SYSTEM CODEC_TEST (* Data Encoding/Decoding Test *)
  (* Standard: 61499 Feasibility Demo *)
  (* Version 0.9, 2006-03-04, JHC, Holobloc Inc, Adjusted frame sizes for Windows XP. *)
  (* Version 0.8, 2006-03-02, JHC, Holobloc Inc, Inserted delay in MONITOR initialization. *)
  (* Version 0.7, 2004-08-04, JHC, Rockwell Automation, Adjusted field sizes for Swing components. *)
  (* Version 0.6, 2001-06-01, JHC, Rockwell Automation, Changed to new IN_ANY, OUT_ANY. *)
  (* Version 0.5, 2001-05-24, JHC, Rockwell Automation, Added applications. *)
  (* Version 0.4, 2001-05-23, JHC, Rockwell Automation, Corrected UDP addresses *)
  (* Version 0.3, 2001-05-18, JHC, Rockwell Automation, Adjusted layouts *)
  (* Version 0.2, 2000-12-09, JHC, Rockwell Automation, Adjusted window heights *)
  (* Version 0.1, 2000-05-16, JHC, Rockwell Automation, File type changed to ".sys" *)
  (* Version 0.0, 2000-04-21, JHC, Rockwell Automation *)
  APPLICATION TEST_BITS (* Test bit string data types *)
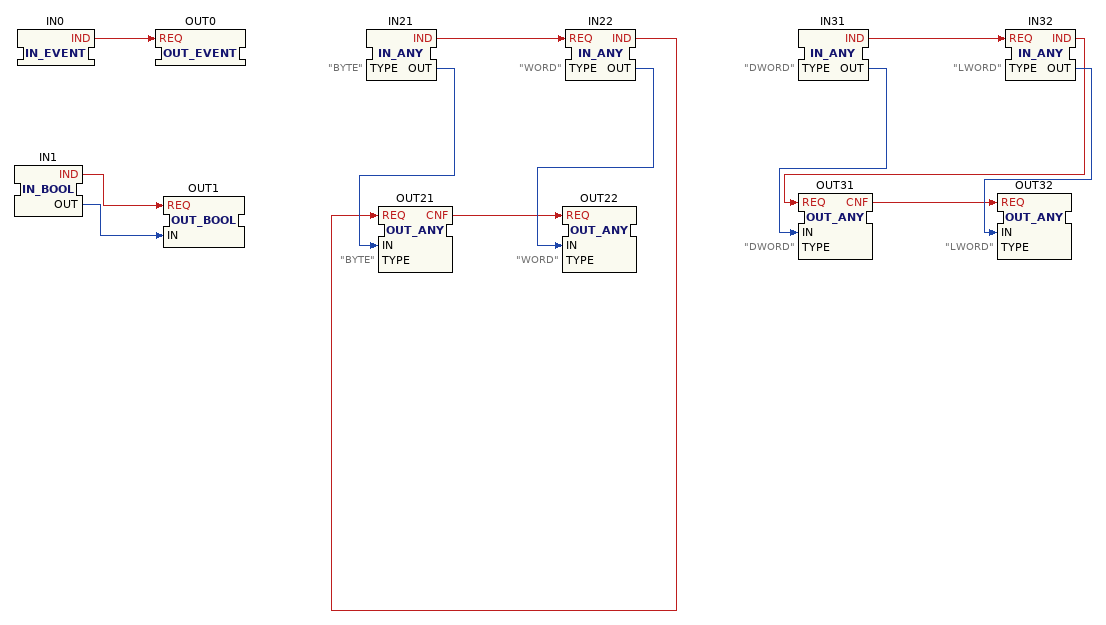
    FBS
      IN0 : IN_EVENT;
      OUT0 : OUT_EVENT;
      IN1 : IN_BOOL;
      OUT1 : OUT_BOOL;
      IN21 : IN_ANY(TYPE := "BYTE");
      OUT21 : OUT_ANY(TYPE := "BYTE");
      IN22 : IN_ANY(TYPE := "WORD");
      OUT22 : OUT_ANY(TYPE := "WORD");
      IN31 : IN_ANY(TYPE := "DWORD");
      OUT31 : OUT_ANY(TYPE := "DWORD");
      IN32 : IN_ANY(TYPE := "LWORD");
      OUT32 : OUT_ANY(TYPE := "LWORD");
    END_FBS
    EVENT_CONNECTIONS
      IN0.IND TO OUT0.REQ;
      IN1.IND TO OUT1.REQ;
      IN21.IND TO IN22.REQ;
      IN22.IND TO OUT21.REQ;
      OUT21.CNF TO OUT22.REQ;
      IN31.IND TO IN32.REQ;
      IN32.IND TO OUT31.REQ;
      OUT31.CNF TO OUT32.REQ;
    END_CONNECTIONS
    DATA_CONNECTIONS
      IN1.OUT TO OUT1.IN;
      IN21.OUT TO OUT21.IN;
      IN22.OUT TO OUT22.IN;
      IN31.OUT TO OUT31.IN;
      IN32.OUT TO OUT32.IN;
    END_CONNECTIONS
  END_APPLICATION
  APPLICATION TEST_INTS (* Test integer data types *)
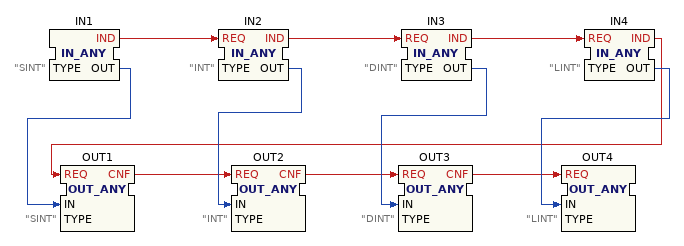
    FBS
      IN1 : IN_ANY(TYPE := "SINT");
      IN2 : IN_ANY(TYPE := "INT");
      IN3 : IN_ANY(TYPE := "DINT");
      IN4 : IN_ANY(TYPE := "LINT");
      OUT1 : OUT_ANY(TYPE := "SINT");
      OUT2 : OUT_ANY(TYPE := "INT");
      OUT3 : OUT_ANY(TYPE := "DINT");
      OUT4 : OUT_ANY(TYPE := "LINT");
    END_FBS
    EVENT_CONNECTIONS
      IN1.IND TO IN2.REQ;
      IN2.IND TO IN3.REQ;
      IN3.IND TO IN4.REQ;
      IN4.IND TO OUT1.REQ;
      OUT1.CNF TO OUT2.REQ;
      OUT2.CNF TO OUT3.REQ;
      OUT3.CNF TO OUT4.REQ;
    END_CONNECTIONS
    DATA_CONNECTIONS
      IN1.OUT TO OUT1.IN;
      IN2.OUT TO OUT2.IN;
      IN3.OUT TO OUT3.IN;
      IN4.OUT TO OUT4.IN;
    END_CONNECTIONS
  END_APPLICATION
  APPLICATION TEST_UINTS (* Test unsigned integer data types *)
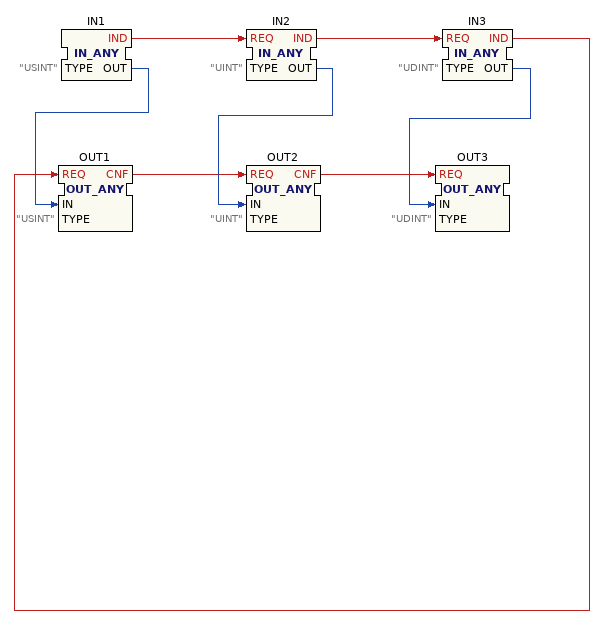
    FBS
      IN1 : IN_ANY(TYPE := "USINT");
      IN2 : IN_ANY(TYPE := "UINT");
      IN3 : IN_ANY(TYPE := "UDINT");
      OUT1 : OUT_ANY(TYPE := "USINT");
      OUT2 : OUT_ANY(TYPE := "UINT");
      OUT3 : OUT_ANY(TYPE := "UDINT");
    END_FBS
    EVENT_CONNECTIONS
      IN1.IND TO IN2.REQ;
      IN2.IND TO IN3.REQ;
      IN3.IND TO OUT1.REQ;
      OUT1.CNF TO OUT2.REQ;
      OUT2.CNF TO OUT3.REQ;
    END_CONNECTIONS
    DATA_CONNECTIONS
      IN1.OUT TO OUT1.IN;
      IN2.OUT TO OUT2.IN;
      IN3.OUT TO OUT3.IN;
    END_CONNECTIONS
  END_APPLICATION
  APPLICATION TEST_REALS (* Test floating point data types *)
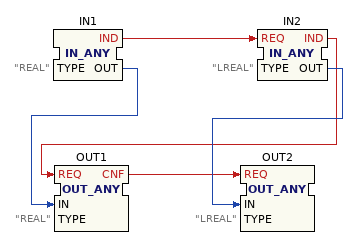
    FBS
      IN1 : IN_ANY(TYPE := "REAL");
      IN2 : IN_ANY(TYPE := "LREAL");
      OUT1 : OUT_ANY(TYPE := "REAL");
      OUT2 : OUT_ANY(TYPE := "LREAL");
    END_FBS
    EVENT_CONNECTIONS
      IN1.IND TO IN2.REQ;
      IN2.IND TO OUT1.REQ;
      OUT1.CNF TO OUT2.REQ;
    END_CONNECTIONS
    DATA_CONNECTIONS
      IN1.OUT TO OUT1.IN;
      IN2.OUT TO OUT2.IN;
    END_CONNECTIONS
  END_APPLICATION
  APPLICATION TEST_TIMES (* Test time data types *)
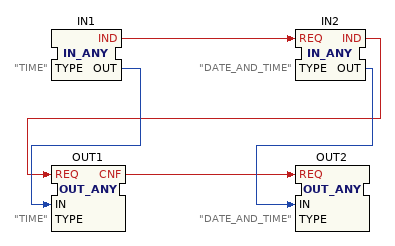
    FBS
      IN1 : IN_ANY(TYPE := "TIME");
      IN2 : IN_ANY(TYPE := "DATE_AND_TIME");
      OUT1 : OUT_ANY(TYPE := "TIME");
      OUT2 : OUT_ANY(TYPE := "DATE_AND_TIME");
    END_FBS
    EVENT_CONNECTIONS
      IN1.IND TO IN2.REQ;
      IN2.IND TO OUT1.REQ;
      OUT1.CNF TO OUT2.REQ;
    END_CONNECTIONS
    DATA_CONNECTIONS
      IN1.OUT TO OUT1.IN;
      IN2.OUT TO OUT2.IN;
    END_CONNECTIONS
  END_APPLICATION
  APPLICATION TEST_STRINGS (* Test string data types *)
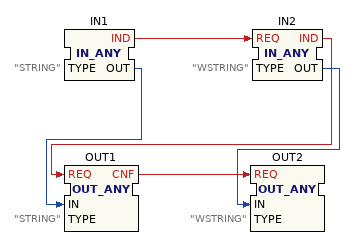
    FBS
      IN1 : IN_ANY(TYPE := "STRING");
      IN2 : IN_ANY(TYPE := "WSTRING");
      OUT1 : OUT_ANY(TYPE := "STRING");
      OUT2 : OUT_ANY(TYPE := "WSTRING");
    END_FBS
    EVENT_CONNECTIONS
      IN1.IND TO IN2.REQ;
      IN2.IND TO OUT1.REQ;
      OUT1.CNF TO OUT2.REQ;
    END_CONNECTIONS
    DATA_CONNECTIONS
      IN1.OUT TO OUT1.IN;
      IN2.OUT TO OUT2.IN;
    END_CONNECTIONS
  END_APPLICATION
  APPLICATION TEST_ARRAY (* Test ARRAYs *)
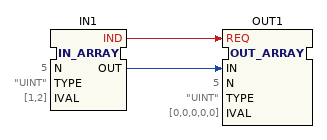
    FBS
      IN1 : IN_ARRAY(N := 5, TYPE := "UINT", IVAL := [1,2]);
      OUT1 : OUT_ARRAY(N := 5, TYPE := "UINT", IVAL := [0,0,0,0,0]);
    END_FBS
    EVENT_CONNECTIONS
      IN1.IND TO OUT1.REQ;
    END_CONNECTIONS
    DATA_CONNECTIONS
      IN1.OUT TO OUT1.IN;
    END_CONNECTIONS
  END_APPLICATION
  APPLICATION TEST_COLOR (* Test  COLOR - Just for fun! *)
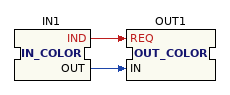
    FBS
      IN1 : IN_COLOR;
      OUT1 : OUT_COLOR;
    END_FBS
    EVENT_CONNECTIONS
      IN1.IND TO OUT1.REQ;
    END_CONNECTIONS
    DATA_CONNECTIONS
      IN1.OUT TO OUT1.IN;
    END_CONNECTIONS
  END_APPLICATION
  DEVICE SEND_BITS : FRAME_DEVICE(BOUNDS := [50,50,175,195], GRID := [1,1])
    RESOURCE RES0 : PANEL_RESOURCE
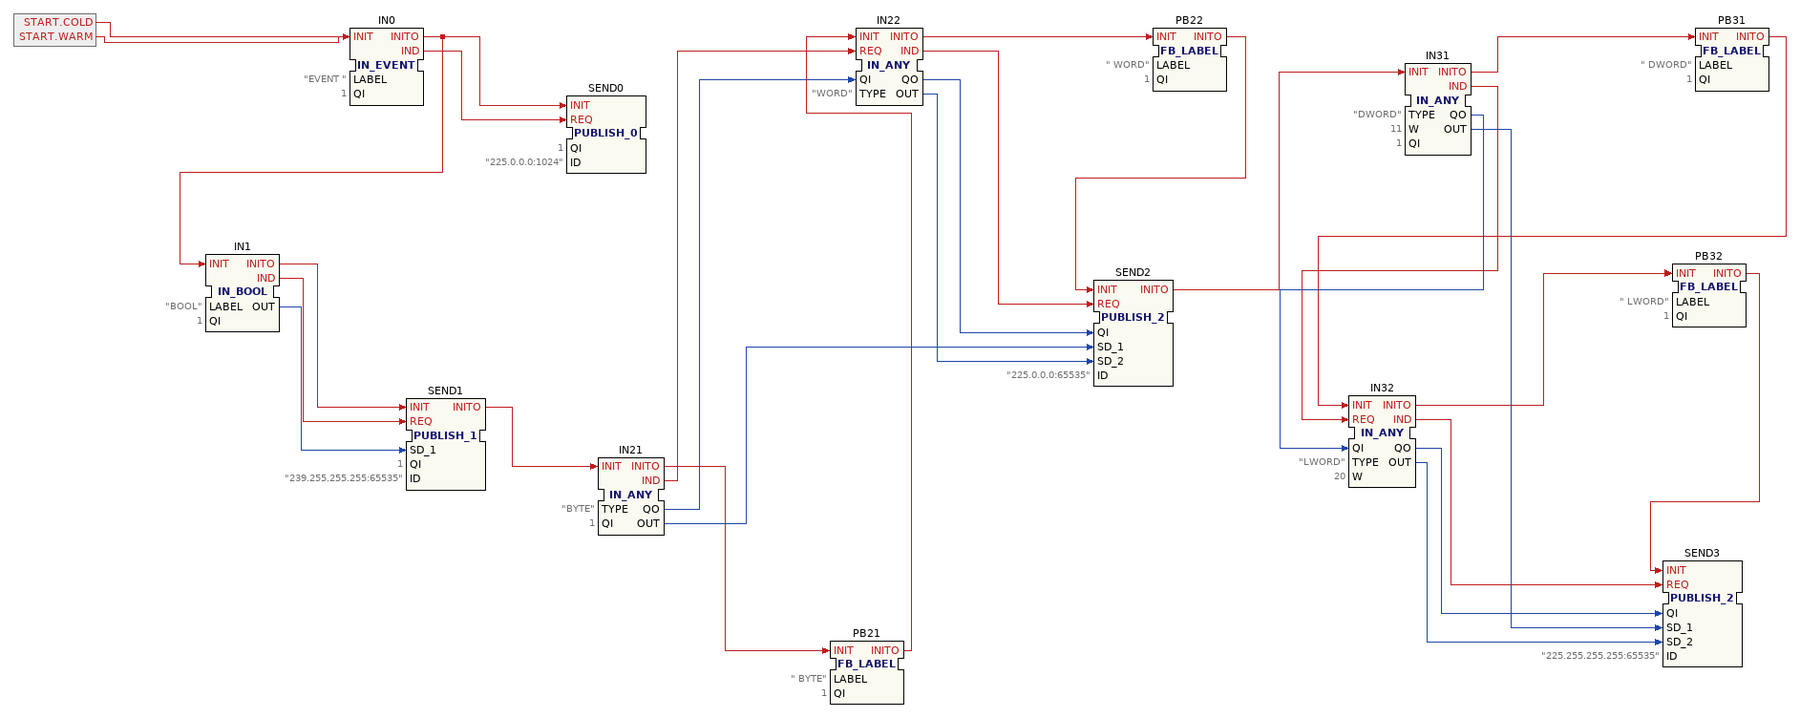
      FBS
        IN0 : IN_EVENT(LABEL := "EVENT   ", QI := 1);
        SEND0 : PUBLISH_0(QI := 1, ID := "225.0.0.0:1024");
        IN1 : IN_BOOL(LABEL := "BOOL", QI := 1);
        SEND1 : PUBLISH_1(QI := 1, ID := "239.255.255.255:65535");
        PB21 : FB_LABEL(LABEL := " BYTE", QI := 1);
        IN21 : IN_ANY(TYPE := "BYTE", QI := 1);
        PB22 : FB_LABEL(LABEL := " WORD", QI := 1);
        IN22 : IN_ANY(TYPE := "WORD");
        SEND2 : PUBLISH_2(ID := "225.0.0.0:65535");
        PB31 : FB_LABEL(LABEL := " DWORD", QI := 1);
        IN31 : IN_ANY(TYPE := "DWORD", W := 11, QI := 1);
        PB32 : FB_LABEL(LABEL := " LWORD", QI := 1);
        IN32 : IN_ANY(TYPE := "LWORD", W := 20);
        SEND3 : PUBLISH_2(ID := "225.255.255.255:65535");
      END_FBS
      EVENT_CONNECTIONS
        START.COLD TO IN0.INIT;
        START.WARM TO IN0.INIT;
        IN0.INITO TO SEND0.INIT;
        IN0.INITO TO IN1.INIT;
        IN1.INITO TO SEND1.INIT;
        SEND1.INITO TO IN21.INIT;
        IN21.INITO TO PB21.INIT;
        PB21.INITO TO IN22.INIT;
        IN22.INITO TO PB22.INIT;
        PB22.INITO TO SEND2.INIT;
        SEND2.INITO TO IN31.INIT;
        IN31.INITO TO PB31.INIT;
        PB31.INITO TO IN32.INIT;
        IN32.INITO TO PB32.INIT;
        PB32.INITO TO SEND3.INIT;
        IN0.IND TO SEND0.REQ;
        IN1.IND TO SEND1.REQ;
        IN21.IND TO IN22.REQ;
        IN22.IND TO SEND2.REQ;
        IN31.IND TO IN32.REQ;
        IN32.IND TO SEND3.REQ;
      END_CONNECTIONS
      DATA_CONNECTIONS
        IN21.QO TO IN22.QI;
        IN22.QO TO SEND2.QI;
        IN31.QO TO IN32.QI;
        IN32.QO TO SEND3.QI;
        IN1.OUT TO SEND1.SD_1;
        IN21.OUT TO SEND2.SD_1;
        IN22.OUT TO SEND2.SD_2;
        IN31.OUT TO SEND3.SD_1;
        IN32.OUT TO SEND3.SD_2;
      END_CONNECTIONS
    END_RESOURCE
  END_DEVICE
  DEVICE RCV_BITS : FRAME_DEVICE(BOUNDS := [225,50,175,195], GRID := [1,1])
    RESOURCE RES0 : PANEL_RESOURCE
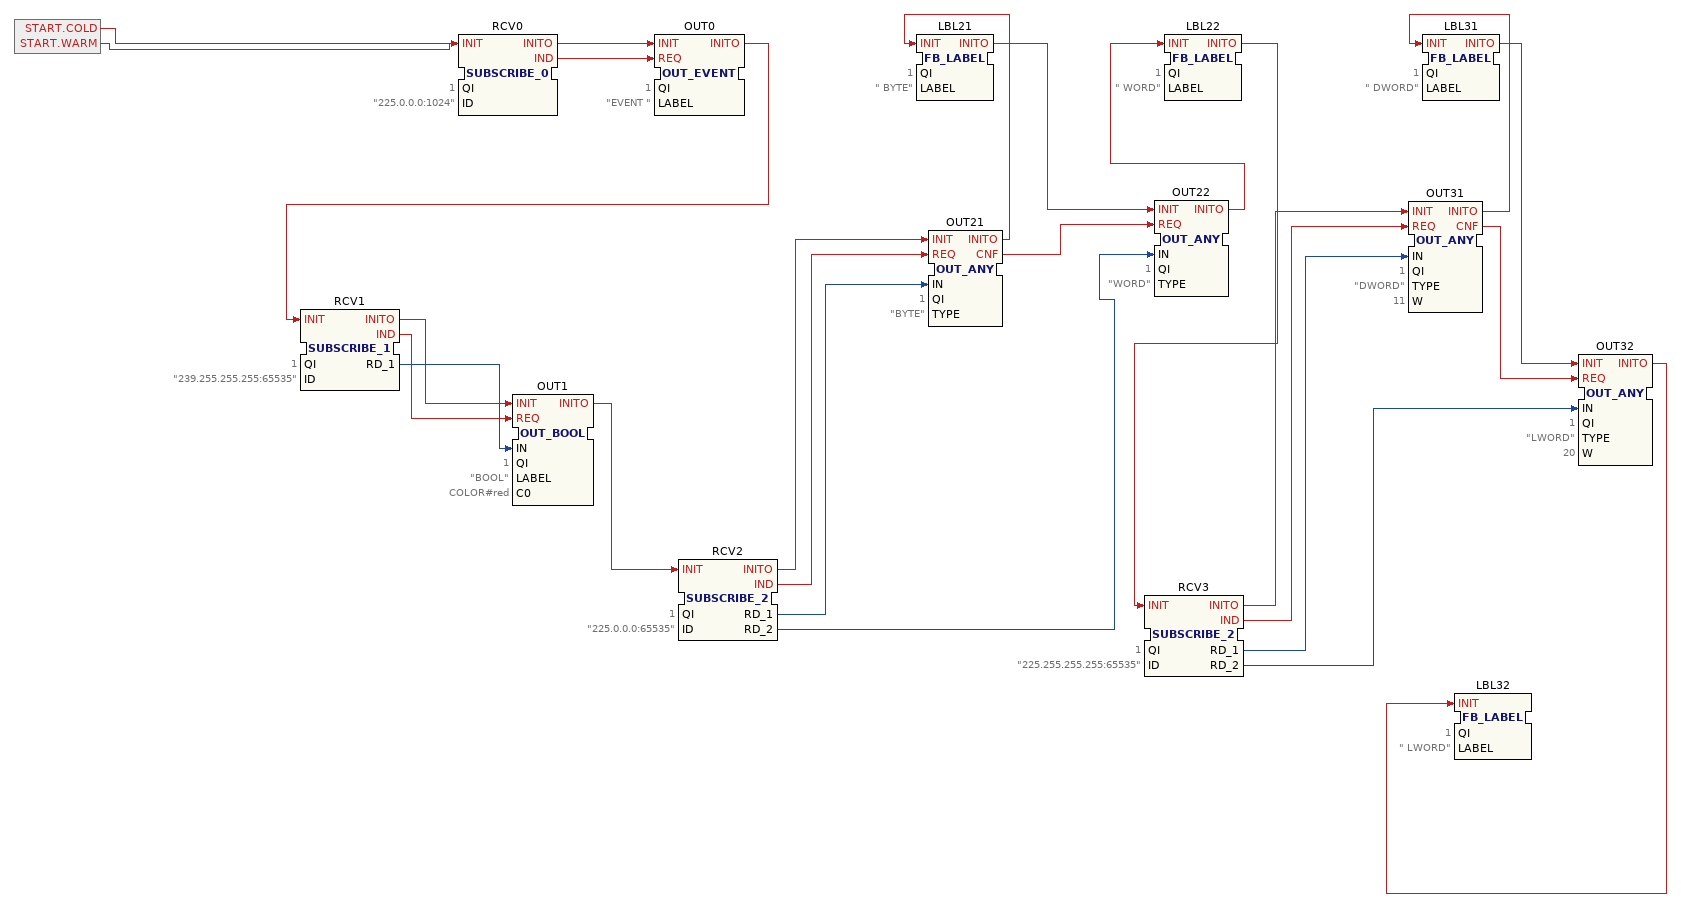
      FBS
        RCV0 : SUBSCRIBE_0(QI := 1, ID := "225.0.0.0:1024");
        OUT0 : OUT_EVENT(QI := 1, LABEL := "EVENT   ");
        RCV1 : SUBSCRIBE_1(QI := 1, ID := "239.255.255.255:65535");
        OUT1 : OUT_BOOL(QI := 1, LABEL := "BOOL", C0 := COLOR#red);
        RCV2 : SUBSCRIBE_2(QI := 1, ID := "225.0.0.0:65535");
        LBL21 : FB_LABEL(QI := 1, LABEL := " BYTE");
        OUT21 : OUT_ANY(QI := 1, TYPE := "BYTE");
        LBL22 : FB_LABEL(QI := 1, LABEL := " WORD");
        OUT22 : OUT_ANY(QI := 1, TYPE := "WORD");
        RCV3 : SUBSCRIBE_2(QI := 1, ID := "225.255.255.255:65535");
        LBL31 : FB_LABEL(QI := 1, LABEL := " DWORD");
        OUT31 : OUT_ANY(QI := 1, TYPE := "DWORD", W := 11);
        LBL32 : FB_LABEL(QI := 1, LABEL := " LWORD");
        OUT32 : OUT_ANY(QI := 1, TYPE := "LWORD", W := 20);
      END_FBS
      EVENT_CONNECTIONS
        START.COLD TO RCV0.INIT;
        START.WARM TO RCV0.INIT;
        RCV0.INITO TO OUT0.INIT;
        OUT0.INITO TO RCV1.INIT;
        RCV1.INITO TO OUT1.INIT;
        OUT1.INITO TO RCV2.INIT;
        RCV2.INITO TO OUT21.INIT;
        OUT21.INITO TO LBL21.INIT;
        LBL21.INITO TO OUT22.INIT;
        OUT22.INITO TO LBL22.INIT;
        LBL22.INITO TO RCV3.INIT;
        RCV3.INITO TO OUT31.INIT;
        OUT31.INITO TO LBL31.INIT;
        LBL31.INITO TO OUT32.INIT;
        OUT32.INITO TO LBL32.INIT;
        RCV0.IND TO OUT0.REQ;
        RCV1.IND TO OUT1.REQ;
        RCV2.IND TO OUT21.REQ;
        OUT21.CNF TO OUT22.REQ;
        RCV3.IND TO OUT31.REQ;
        OUT31.CNF TO OUT32.REQ;
      END_CONNECTIONS
      DATA_CONNECTIONS
        RCV1.RD_1 TO OUT1.IN;
        RCV2.RD_1 TO OUT21.IN;
        RCV2.RD_2 TO OUT22.IN;
        RCV3.RD_1 TO OUT31.IN;
        RCV3.RD_2 TO OUT32.IN;
      END_CONNECTIONS
    END_RESOURCE
  END_DEVICE
  DEVICE SEND_INTS : FRAME_DEVICE(BOUNDS := [50,240,175,170], GRID := [1,1])
    RESOURCE RES0 : PANEL_RESOURCE
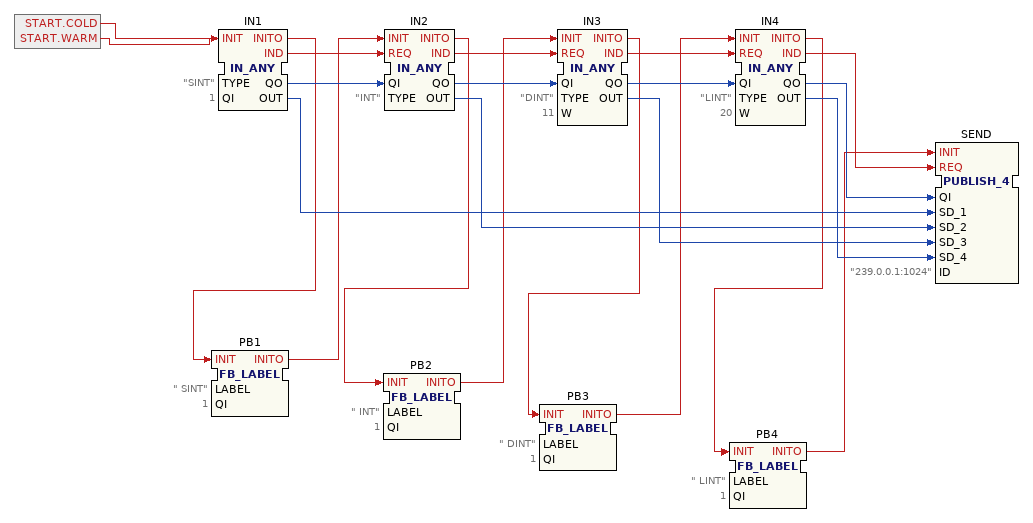
      FBS
        PB1 : FB_LABEL(LABEL := " SINT", QI := 1);
        IN1 : IN_ANY(TYPE := "SINT", QI := 1);
        PB2 : FB_LABEL(LABEL := " INT", QI := 1);
        IN2 : IN_ANY(TYPE := "INT");
        PB3 : FB_LABEL(LABEL := " DINT", QI := 1);
        IN3 : IN_ANY(TYPE := "DINT", W := 11);
        PB4 : FB_LABEL(LABEL := " LINT", QI := 1);
        IN4 : IN_ANY(TYPE := "LINT", W := 20);
        SEND : PUBLISH_4(ID := "239.0.0.1:1024");
      END_FBS
      EVENT_CONNECTIONS
        START.COLD TO IN1.INIT;
        START.WARM TO IN1.INIT;
        IN1.INITO TO PB1.INIT;
        PB1.INITO TO IN2.INIT;
        IN2.INITO TO PB2.INIT;
        PB2.INITO TO IN3.INIT;
        IN3.INITO TO PB3.INIT;
        PB3.INITO TO IN4.INIT;
        IN4.INITO TO PB4.INIT;
        PB4.INITO TO SEND.INIT;
        IN1.IND TO IN2.REQ;
        IN2.IND TO IN3.REQ;
        IN3.IND TO IN4.REQ;
        IN4.IND TO SEND.REQ;
      END_CONNECTIONS
      DATA_CONNECTIONS
        IN1.QO TO IN2.QI;
        IN2.QO TO IN3.QI;
        IN3.QO TO IN4.QI;
        IN4.QO TO SEND.QI;
        IN1.OUT TO SEND.SD_1;
        IN2.OUT TO SEND.SD_2;
        IN3.OUT TO SEND.SD_3;
        IN4.OUT TO SEND.SD_4;
      END_CONNECTIONS
    END_RESOURCE
  END_DEVICE
  DEVICE RCV_INTS : FRAME_DEVICE(BOUNDS := [225,240,175,170], GRID := [1,1])
    RESOURCE RES0 : PANEL_RESOURCE
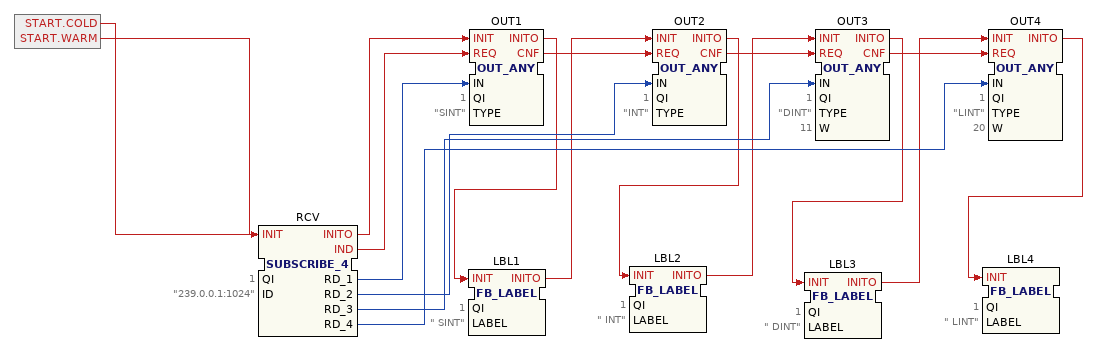
      FBS
        RCV : SUBSCRIBE_4(QI := 1, ID := "239.0.0.1:1024");
        LBL1 : FB_LABEL(QI := 1, LABEL := " SINT");
        OUT1 : OUT_ANY(QI := 1, TYPE := "SINT");
        LBL2 : FB_LABEL(QI := 1, LABEL := " INT");
        OUT2 : OUT_ANY(QI := 1, TYPE := "INT");
        LBL3 : FB_LABEL(QI := 1, LABEL := " DINT");
        OUT3 : OUT_ANY(QI := 1, TYPE := "DINT", W := 11);
        LBL4 : FB_LABEL(QI := 1, LABEL := " LINT");
        OUT4 : OUT_ANY(QI := 1, TYPE := "LINT", W := 20);
      END_FBS
      EVENT_CONNECTIONS
        START.COLD TO RCV.INIT;
        START.WARM TO RCV.INIT;
        RCV.INITO TO OUT1.INIT;
        OUT1.INITO TO LBL1.INIT;
        LBL1.INITO TO OUT2.INIT;
        OUT2.INITO TO LBL2.INIT;
        LBL2.INITO TO OUT3.INIT;
        OUT3.INITO TO LBL3.INIT;
        LBL3.INITO TO OUT4.INIT;
        OUT4.INITO TO LBL4.INIT;
        RCV.IND TO OUT1.REQ;
        OUT1.CNF TO OUT2.REQ;
        OUT2.CNF TO OUT3.REQ;
        OUT3.CNF TO OUT4.REQ;
      END_CONNECTIONS
      DATA_CONNECTIONS
        RCV.RD_1 TO OUT1.IN;
        RCV.RD_2 TO OUT2.IN;
        RCV.RD_3 TO OUT3.IN;
        RCV.RD_4 TO OUT4.IN;
      END_CONNECTIONS
    END_RESOURCE
  END_DEVICE
  DEVICE SEND_UINTS : FRAME_DEVICE(BOUNDS := [50,405,175,120], GRID := [1,1])
    RESOURCE RES0 : PANEL_RESOURCE
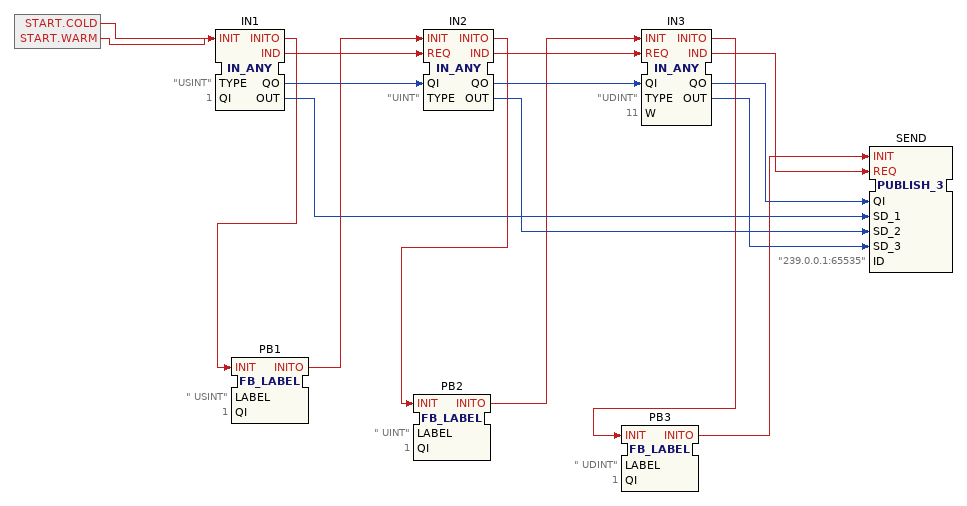
      FBS
        PB1 : FB_LABEL(LABEL := " USINT", QI := 1);
        IN1 : IN_ANY(TYPE := "USINT", QI := 1);
        PB2 : FB_LABEL(LABEL := " UINT", QI := 1);
        IN2 : IN_ANY(TYPE := "UINT");
        PB3 : FB_LABEL(LABEL := " UDINT", QI := 1);
        IN3 : IN_ANY(TYPE := "UDINT", W := 11);
        SEND : PUBLISH_3(ID := "239.0.0.1:65535");
      END_FBS
      EVENT_CONNECTIONS
        START.COLD TO IN1.INIT;
        START.WARM TO IN1.INIT;
        IN1.INITO TO PB1.INIT;
        PB1.INITO TO IN2.INIT;
        IN2.INITO TO PB2.INIT;
        PB2.INITO TO IN3.INIT;
        IN3.INITO TO PB3.INIT;
        PB3.INITO TO SEND.INIT;
        IN1.IND TO IN2.REQ;
        IN2.IND TO IN3.REQ;
        IN3.IND TO SEND.REQ;
      END_CONNECTIONS
      DATA_CONNECTIONS
        IN1.QO TO IN2.QI;
        IN2.QO TO IN3.QI;
        IN3.QO TO SEND.QI;
        IN1.OUT TO SEND.SD_1;
        IN2.OUT TO SEND.SD_2;
        IN3.OUT TO SEND.SD_3;
      END_CONNECTIONS
    END_RESOURCE
  END_DEVICE
  DEVICE RCV_UINTS : FRAME_DEVICE(BOUNDS := [225,405,175,120], GRID := [1,1])
    RESOURCE RES0 : PANEL_RESOURCE
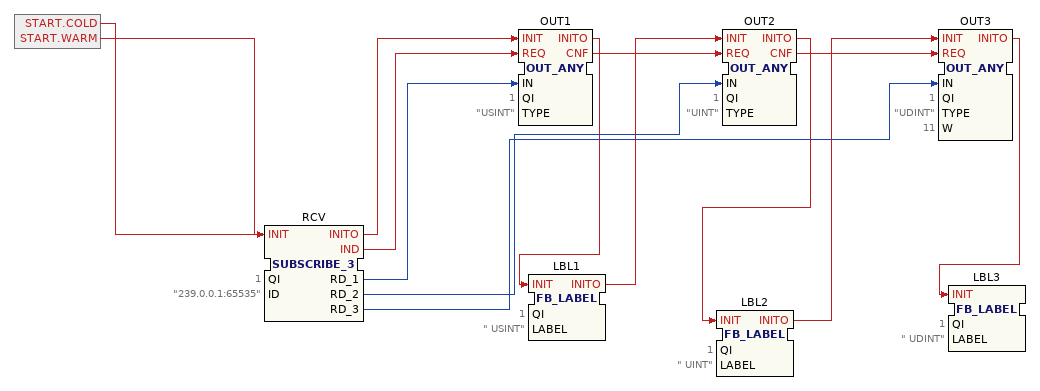
      FBS
        RCV : SUBSCRIBE_3(QI := 1, ID := "239.0.0.1:65535");
        LBL1 : FB_LABEL(QI := 1, LABEL := " USINT");
        OUT1 : OUT_ANY(QI := 1, TYPE := "USINT");
        LBL2 : FB_LABEL(QI := 1, LABEL := " UINT");
        OUT2 : OUT_ANY(QI := 1, TYPE := "UINT");
        LBL3 : FB_LABEL(QI := 1, LABEL := " UDINT");
        OUT3 : OUT_ANY(QI := 1, TYPE := "UDINT", W := 11);
      END_FBS
      EVENT_CONNECTIONS
        START.COLD TO RCV.INIT;
        START.WARM TO RCV.INIT;
        RCV.INITO TO OUT1.INIT;
        OUT1.INITO TO LBL1.INIT;
        LBL1.INITO TO OUT2.INIT;
        OUT2.INITO TO LBL2.INIT;
        LBL2.INITO TO OUT3.INIT;
        OUT3.INITO TO LBL3.INIT;
        RCV.IND TO OUT1.REQ;
        OUT1.CNF TO OUT2.REQ;
        OUT2.CNF TO OUT3.REQ;
      END_CONNECTIONS
      DATA_CONNECTIONS
        RCV.RD_1 TO OUT1.IN;
        RCV.RD_2 TO OUT2.IN;
        RCV.RD_3 TO OUT3.IN;
      END_CONNECTIONS
    END_RESOURCE
  END_DEVICE
  DEVICE SEND_REALS : FRAME_DEVICE(BOUNDS := [50,520,175,100], GRID := [1,1])
    RESOURCE RES0 : PANEL_RESOURCE
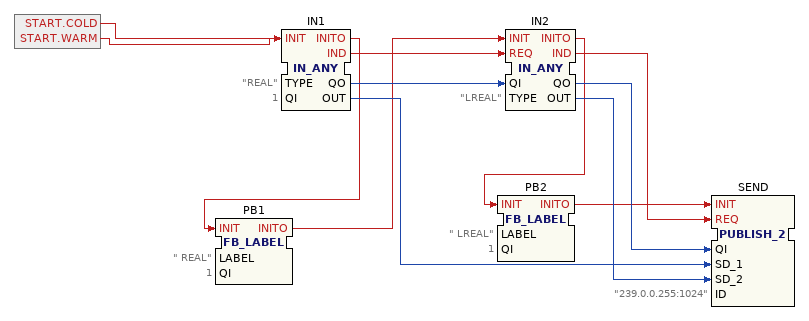
      FBS
        PB1 : FB_LABEL(LABEL := " REAL", QI := 1);
        IN1 : IN_ANY(TYPE := "REAL", QI := 1);
        PB2 : FB_LABEL(LABEL := " LREAL", QI := 1);
        IN2 : IN_ANY(TYPE := "LREAL");
        SEND : PUBLISH_2(ID := "239.0.0.255:1024");
      END_FBS
      EVENT_CONNECTIONS
        START.COLD TO IN1.INIT;
        START.WARM TO IN1.INIT;
        IN1.INITO TO PB1.INIT;
        PB1.INITO TO IN2.INIT;
        IN2.INITO TO PB2.INIT;
        PB2.INITO TO SEND.INIT;
        IN1.IND TO IN2.REQ;
        IN2.IND TO SEND.REQ;
      END_CONNECTIONS
      DATA_CONNECTIONS
        IN1.QO TO IN2.QI;
        IN2.QO TO SEND.QI;
        IN1.OUT TO SEND.SD_1;
        IN2.OUT TO SEND.SD_2;
      END_CONNECTIONS
    END_RESOURCE
  END_DEVICE
  DEVICE RCV_REALS : FRAME_DEVICE(BOUNDS := [225,520,175,100], GRID := [1,1])
    RESOURCE RES0 : PANEL_RESOURCE
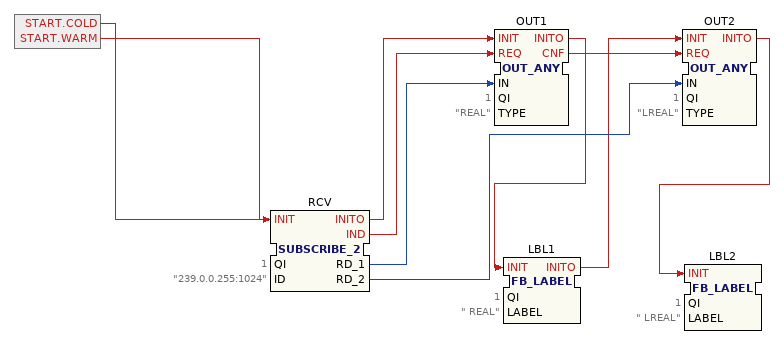
      FBS
        RCV : SUBSCRIBE_2(QI := 1, ID := "239.0.0.255:1024");
        LBL1 : FB_LABEL(QI := 1, LABEL := " REAL");
        OUT1 : OUT_ANY(QI := 1, TYPE := "REAL");
        LBL2 : FB_LABEL(QI := 1, LABEL := " LREAL");
        OUT2 : OUT_ANY(QI := 1, TYPE := "LREAL");
      END_FBS
      EVENT_CONNECTIONS
        START.COLD TO RCV.INIT;
        START.WARM TO RCV.INIT;
        RCV.INITO TO OUT1.INIT;
        OUT1.INITO TO LBL1.INIT;
        LBL1.INITO TO OUT2.INIT;
        OUT2.INITO TO LBL2.INIT;
        RCV.IND TO OUT1.REQ;
        OUT1.CNF TO OUT2.REQ;
      END_CONNECTIONS
      DATA_CONNECTIONS
        RCV.RD_1 TO OUT1.IN;
        RCV.RD_2 TO OUT2.IN;
      END_CONNECTIONS
    END_RESOURCE
  END_DEVICE
  DEVICE MONITOR : FRAME_DEVICE(BOUNDS := [400,50,400,225], GRID := [1,1])
    RESOURCE RES0 : PANEL_RESOURCE
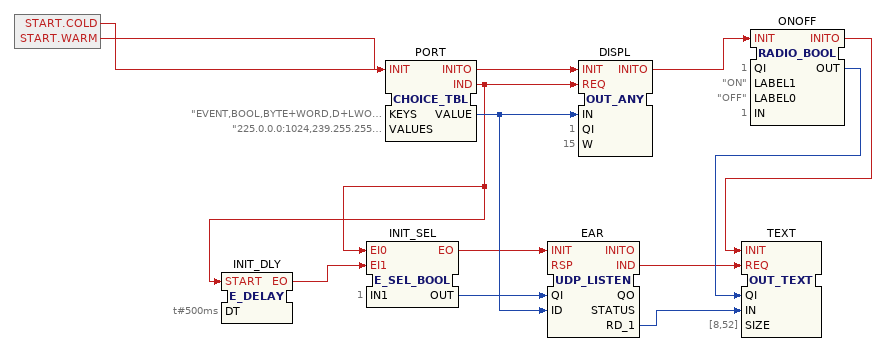
      FBS
        PORT : CHOICE_TBL(KEYS := "EVENT,BOOL,BYTE+WORD,D+LWORD,INTS,UINTS,REALS,TIMES,STRINGS,ARRAYS,COLOR", VALUES := "225.0.0.0:1024,239.255.255.255:65535,225.0.0.0:65535,225.255.255.255:65535,239.0.0.1:1024,239.0.0.1:65535,239.0.0.255:1024,239.0.0.255:65535,239.0.255.255:1024,239.0.255.255:65535,239.255.255.255:1024");
        DISPL : OUT_ANY(QI := 1, W := 15);
        EAR : UDP_LISTEN;
        ONOFF : RADIO_BOOL(QI := 1, LABEL1 := "ON", LABEL0 := "OFF", IN := 1);
        TEXT : OUT_TEXT(SIZE := [8,52]);
        INIT_SEL : E_SEL_BOOL(IN1 := 1);
        INIT_DLY : E_DELAY(DT := t#500ms);
      END_FBS
      EVENT_CONNECTIONS
        START.COLD TO PORT.INIT;
        START.WARM TO PORT.INIT;
        PORT.INITO TO DISPL.INIT;
        DISPL.INITO TO ONOFF.INIT;
        ONOFF.INITO TO TEXT.INIT;
        PORT.IND TO DISPL.REQ;
        EAR.IND TO TEXT.REQ;
        PORT.IND TO INIT_SEL.EI0;
        INIT_SEL.EO TO EAR.INIT;
        INIT_DLY.EO TO INIT_SEL.EI1;
        PORT.IND TO INIT_DLY.START;
      END_CONNECTIONS
      DATA_CONNECTIONS
        PORT.VALUE TO DISPL.IN;
        PORT.VALUE TO EAR.ID;
        ONOFF.OUT TO TEXT.QI;
        EAR.RD_1 TO TEXT.IN;
        INIT_SEL.OUT TO EAR.QI;
      END_CONNECTIONS
    END_RESOURCE
  END_DEVICE
  DEVICE SEND_TIMES : FRAME_DEVICE(BOUNDS := [400,270,200,115], GRID := [1,1])
    RESOURCE RES0 : PANEL_RESOURCE
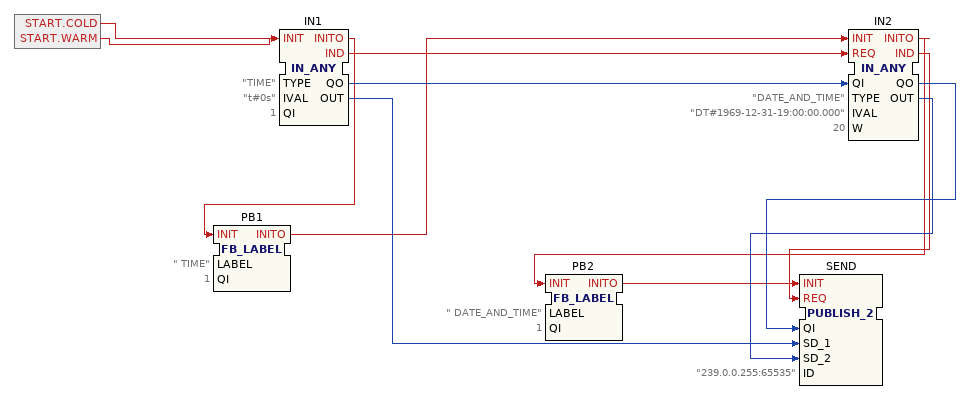
      FBS
        PB1 : FB_LABEL(LABEL := " TIME", QI := 1);
        IN1 : IN_ANY(TYPE := "TIME", IVAL := "t#0s", QI := 1);
        PB2 : FB_LABEL(LABEL := " DATE_AND_TIME", QI := 1);
        IN2 : IN_ANY(TYPE := "DATE_AND_TIME", IVAL := "DT#1969-12-31-19:00:00.000", W := 20);
        SEND : PUBLISH_2(ID := "239.0.0.255:65535");
      END_FBS
      EVENT_CONNECTIONS
        START.COLD TO IN1.INIT;
        START.WARM TO IN1.INIT;
        IN1.INITO TO PB1.INIT;
        PB1.INITO TO IN2.INIT;
        IN2.INITO TO PB2.INIT;
        PB2.INITO TO SEND.INIT;
        IN1.IND TO IN2.REQ;
        IN2.IND TO SEND.REQ;
      END_CONNECTIONS
      DATA_CONNECTIONS
        IN1.QO TO IN2.QI;
        IN2.QO TO SEND.QI;
        IN1.OUT TO SEND.SD_1;
        IN2.OUT TO SEND.SD_2;
      END_CONNECTIONS
    END_RESOURCE
  END_DEVICE
  DEVICE RCV_TIMES : FRAME_DEVICE(BOUNDS := [600,270,200,115], GRID := [1,1])
    RESOURCE RES0 : PANEL_RESOURCE
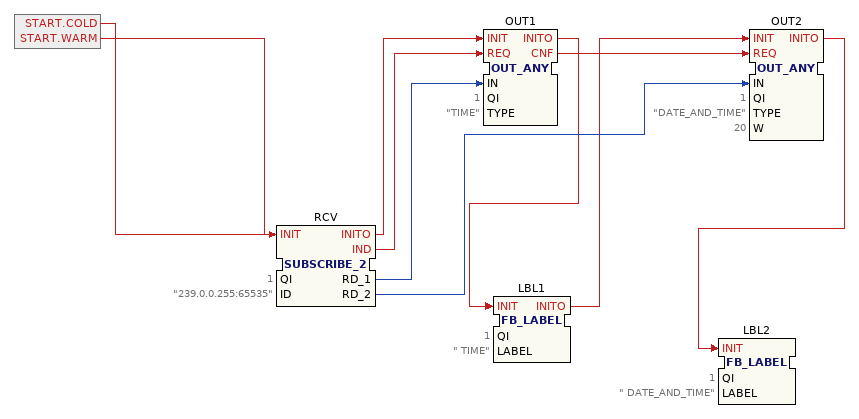
      FBS
        RCV : SUBSCRIBE_2(QI := 1, ID := "239.0.0.255:65535");
        LBL1 : FB_LABEL(QI := 1, LABEL := " TIME");
        OUT1 : OUT_ANY(QI := 1, TYPE := "TIME");
        LBL2 : FB_LABEL(QI := 1, LABEL := " DATE_AND_TIME");
        OUT2 : OUT_ANY(QI := 1, TYPE := "DATE_AND_TIME", W := 20);
      END_FBS
      EVENT_CONNECTIONS
        START.COLD TO RCV.INIT;
        START.WARM TO RCV.INIT;
        RCV.INITO TO OUT1.INIT;
        OUT1.INITO TO LBL1.INIT;
        LBL1.INITO TO OUT2.INIT;
        OUT2.INITO TO LBL2.INIT;
        RCV.IND TO OUT1.REQ;
        OUT1.CNF TO OUT2.REQ;
      END_CONNECTIONS
      DATA_CONNECTIONS
        RCV.RD_1 TO OUT1.IN;
        RCV.RD_2 TO OUT2.IN;
      END_CONNECTIONS
    END_RESOURCE
  END_DEVICE
  DEVICE SEND_STRINGS : FRAME_DEVICE(BOUNDS := [400,385,200,95], GRID := [1,1])
    RESOURCE RES0 : PANEL_RESOURCE
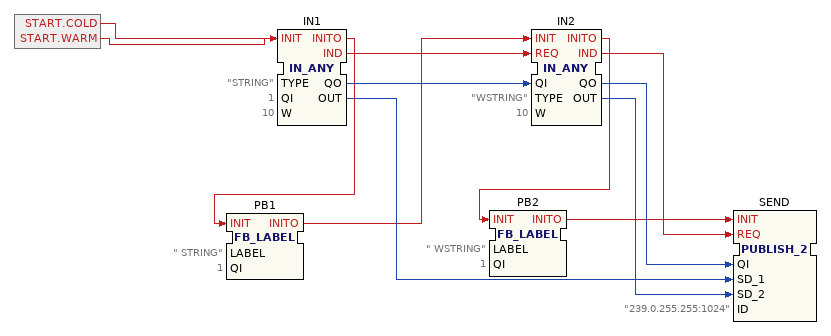
      FBS
        PB1 : FB_LABEL(LABEL := " STRING", QI := 1);
        IN1 : IN_ANY(TYPE := "STRING", QI := 1, W := 10);
        PB2 : FB_LABEL(LABEL := " WSTRING", QI := 1);
        IN2 : IN_ANY(TYPE := "WSTRING", W := 10);
        SEND : PUBLISH_2(ID := "239.0.255.255:1024");
      END_FBS
      EVENT_CONNECTIONS
        START.COLD TO IN1.INIT;
        START.WARM TO IN1.INIT;
        IN1.INITO TO PB1.INIT;
        PB1.INITO TO IN2.INIT;
        IN2.INITO TO PB2.INIT;
        PB2.INITO TO SEND.INIT;
        IN1.IND TO IN2.REQ;
        IN2.IND TO SEND.REQ;
      END_CONNECTIONS
      DATA_CONNECTIONS
        IN1.QO TO IN2.QI;
        IN2.QO TO SEND.QI;
        IN1.OUT TO SEND.SD_1;
        IN2.OUT TO SEND.SD_2;
      END_CONNECTIONS
    END_RESOURCE
  END_DEVICE
  DEVICE RCV_STRINGS : FRAME_DEVICE(BOUNDS := [600,385,200,95], GRID := [1,1])
    RESOURCE RES0 : PANEL_RESOURCE
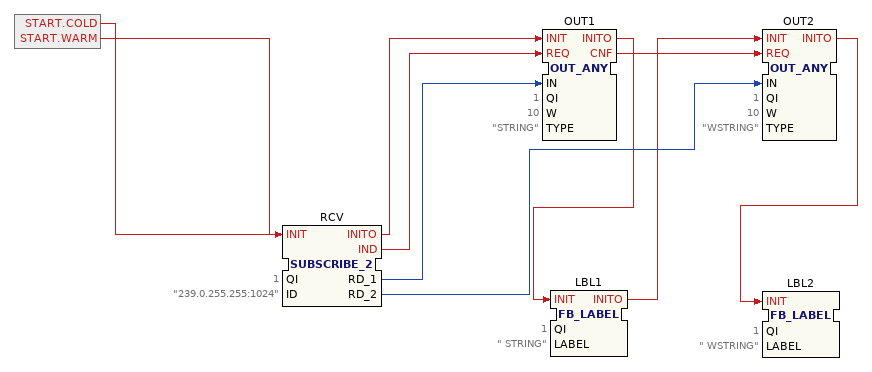
      FBS
        RCV : SUBSCRIBE_2(QI := 1, ID := "239.0.255.255:1024");
        LBL1 : FB_LABEL(QI := 1, LABEL := " STRING");
        OUT1 : OUT_ANY(QI := 1, W := 10, TYPE := "STRING");
        LBL2 : FB_LABEL(QI := 1, LABEL := " WSTRING");
        OUT2 : OUT_ANY(QI := 1, W := 10, TYPE := "WSTRING");
      END_FBS
      EVENT_CONNECTIONS
        START.COLD TO RCV.INIT;
        START.WARM TO RCV.INIT;
        RCV.INITO TO OUT1.INIT;
        OUT1.INITO TO LBL1.INIT;
        LBL1.INITO TO OUT2.INIT;
        OUT2.INITO TO LBL2.INIT;
        RCV.IND TO OUT1.REQ;
        OUT1.CNF TO OUT2.REQ;
      END_CONNECTIONS
      DATA_CONNECTIONS
        RCV.RD_1 TO OUT1.IN;
        RCV.RD_2 TO OUT2.IN;
      END_CONNECTIONS
    END_RESOURCE
  END_DEVICE
  DEVICE SEND_ARRAY : FRAME_DEVICE(BOUNDS := [400,480,210,80], GRID := [1,1])
    RESOURCE RES0 : PANEL_RESOURCE
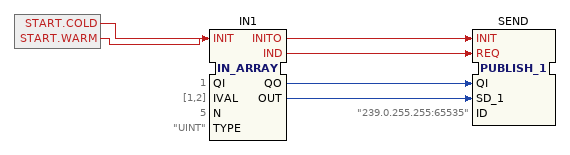
      FBS
        IN1 : IN_ARRAY(QI := 1, IVAL := [1,2], N := 5, TYPE := "UINT");
        SEND : PUBLISH_1(ID := "239.0.255.255:65535");
      END_FBS
      EVENT_CONNECTIONS
        START.COLD TO IN1.INIT;
        START.WARM TO IN1.INIT;
        IN1.INITO TO SEND.INIT;
        IN1.IND TO SEND.REQ;
      END_CONNECTIONS
      DATA_CONNECTIONS
        IN1.QO TO SEND.QI;
        IN1.OUT TO SEND.SD_1;
      END_CONNECTIONS
    END_RESOURCE
  END_DEVICE
  DEVICE RCV_ARRAY : FRAME_DEVICE(BOUNDS := [610,480,190,80], GRID := [1,1])
    RESOURCE RES0 : PANEL_RESOURCE
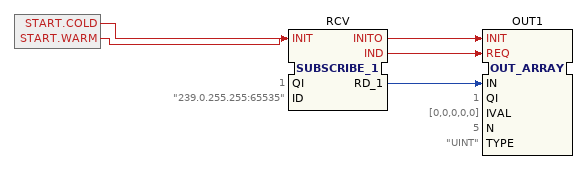
      FBS
        RCV : SUBSCRIBE_1(QI := 1, ID := "239.0.255.255:65535");
        OUT1 : OUT_ARRAY(QI := 1, IVAL := [0,0,0,0,0], N := 5, TYPE := "UINT");
      END_FBS
      EVENT_CONNECTIONS
        START.COLD TO RCV.INIT;
        START.WARM TO RCV.INIT;
        RCV.INITO TO OUT1.INIT;
        RCV.IND TO OUT1.REQ;
      END_CONNECTIONS
      DATA_CONNECTIONS
        RCV.RD_1 TO OUT1.IN;
      END_CONNECTIONS
    END_RESOURCE
  END_DEVICE
  DEVICE SEND_COLOR : FRAME_DEVICE(BOUNDS := [400,560,210,90], GRID := [1,1])
    RESOURCE RES0 : PANEL_RESOURCE
      FBS
        IN1 : IN_COLOR(QI := 1);
        SEND : PUBLISH_1(QI := 1, ID := "239.255.255.255:1024");
      END_FBS
      EVENT_CONNECTIONS
        START.COLD TO IN1.INIT;
        START.WARM TO IN1.INIT;
        IN1.INITO TO SEND.INIT;
        IN1.IND TO SEND.REQ;
      END_CONNECTIONS
      DATA_CONNECTIONS
        IN1.OUT TO SEND.SD_1;
      END_CONNECTIONS
    END_RESOURCE
  END_DEVICE
  DEVICE RCV_COLOR : FRAME_DEVICE(BOUNDS := [610,560,190,90], GRID := [1,1])
    RESOURCE RES0 : PANEL_RESOURCE
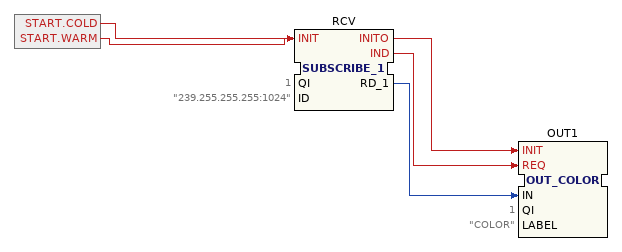
      FBS
        RCV : SUBSCRIBE_1(QI := 1, ID := "239.255.255.255:1024");
        OUT1 : OUT_COLOR(QI := 1, LABEL := "COLOR");
      END_FBS
      EVENT_CONNECTIONS
        START.COLD TO RCV.INIT;
        START.WARM TO RCV.INIT;
        RCV.INITO TO OUT1.INIT;
        RCV.IND TO OUT1.REQ;
      END_CONNECTIONS
      DATA_CONNECTIONS
        RCV.RD_1 TO OUT1.IN;
      END_CONNECTIONS
    END_RESOURCE
  END_DEVICE
  MAPPINGS
    TEST_BITS.IN0 ON SEND_BITS.RES0.IN0;
    TEST_BITS.OUT0 ON RCV_BITS.RES0.OUT0;
    TEST_BITS.IN1 ON SEND_BITS.RES0.IN1;
    TEST_BITS.OUT1 ON RCV_BITS.RES0.OUT1;
    TEST_BITS.PB21 ON SEND_BITS.RES0.PB21;
    TEST_BITS.IN21 ON SEND_BITS.RES0.IN21;
    TEST_BITS.PB22 ON SEND_BITS.RES0.PB22;
    TEST_BITS.OUT21 ON RCV_BITS.RES0.OUT21;
    TEST_BITS.IN22 ON SEND_BITS.RES0.IN22;
    TEST_BITS.OUT22 ON RCV_BITS.RES0.OUT22;
    TEST_BITS.PB31 ON SEND_BITS.RES0.PB31;
    TEST_BITS.IN31 ON SEND_BITS.RES0.IN31;
    TEST_BITS.OUT31 ON RCV_BITS.RES0.OUT31;
    TEST_BITS.PB32 ON SEND_BITS.RES0.PB32;
    TEST_BITS.IN32 ON SEND_BITS.RES0.IN32;
    TEST_BITS.OUT32 ON RCV_BITS.RES0.OUT32;
    TEST_INTS.PB1 ON SEND_INTS.RES0.PB1;
    TEST_INTS.IN1 ON SEND_INTS.RES0.IN1;
    TEST_INTS.PB2 ON SEND_INTS.RES0.PB2;
    TEST_INTS.IN2 ON SEND_INTS.RES0.IN2;
    TEST_INTS.PB3 ON SEND_INTS.RES0.PB3;
    TEST_INTS.IN3 ON SEND_INTS.RES0.IN3;
    TEST_INTS.PB4 ON SEND_INTS.RES0.PB4;
    TEST_INTS.IN4 ON SEND_INTS.RES0.IN4;
    TEST_INTS.OUT1 ON RCV_INTS.RES0.OUT1;
    TEST_INTS.OUT2 ON RCV_INTS.RES0.OUT2;
    TEST_INTS.OUT3 ON RCV_INTS.RES0.OUT3;
    TEST_INTS.OUT4 ON RCV_INTS.RES0.OUT4;
    TEST_UINTS.PB1 ON SEND_UINTS.RES0.PB1;
    TEST_UINTS.IN1 ON SEND_UINTS.RES0.IN1;
    TEST_UINTS.PB2 ON SEND_UINTS.RES0.PB2;
    TEST_UINTS.IN2 ON SEND_UINTS.RES0.IN2;
    TEST_UINTS.PB3 ON SEND_UINTS.RES0.PB3;
    TEST_UINTS.IN3 ON SEND_UINTS.RES0.IN3;
    TEST_UINTS.OUT1 ON RCV_UINTS.RES0.OUT1;
    TEST_UINTS.OUT2 ON RCV_UINTS.RES0.OUT2;
    TEST_UINTS.OUT3 ON RCV_UINTS.RES0.OUT3;
    TEST_REALS.PB1 ON SEND_REALS.RES0.PB1;
    TEST_REALS.IN1 ON SEND_REALS.RES0.IN1;
    TEST_REALS.PB2 ON SEND_REALS.RES0.PB2;
    TEST_REALS.IN2 ON SEND_REALS.RES0.IN2;
    TEST_REALS.OUT1 ON RCV_REALS.RES0.OUT1;
    TEST_REALS.OUT2 ON RCV_REALS.RES0.OUT2;
    TEST_TIMES.PB1 ON SEND_TIMES.RES0.PB1;
    TEST_TIMES.IN1 ON SEND_TIMES.RES0.IN1;
    TEST_TIMES.PB2 ON SEND_TIMES.RES0.PB2;
    TEST_TIMES.IN2 ON SEND_TIMES.RES0.IN2;
    TEST_TIMES.OUT1 ON RCV_TIMES.RES0.OUT1;
    TEST_TIMES.OUT2 ON RCV_TIMES.RES0.OUT2;
    TEST_STRINGS.PB1 ON SEND_STRINGS.RES0.PB1;
    TEST_STRINGS.IN1 ON SEND_STRINGS.RES0.IN1;
    TEST_STRINGS.PB2 ON SEND_STRINGS.RES0.PB2;
    TEST_STRINGS.IN2 ON SEND_STRINGS.RES0.IN2;
    TEST_STRINGS.OUT1 ON RCV_STRINGS.RES0.OUT1;
    TEST_STRINGS.OUT2 ON RCV_STRINGS.RES0.OUT2;
    TEST_ARRAY.PB1 ON SEND_ARRAY.RES0.PB1;
    TEST_ARRAY.IN1 ON SEND_ARRAY.RES0.PB1;
    TEST_ARRAY.OUT1 ON RCV_ARRAY.RES0.OUT1;
    TEST_COLOR.IN1 ON SEND_COLOR.RES0.IN1;
    TEST_COLOR.OUT1 ON RCV_COLOR.RES0.OUT1;
  END_MAPPINGS
END_SYSTEM
